// TIA Portal V20 export
TYPE "OPC_DestRequest_Ack"
// stored: Namespace ProductionLine
   STRUCT
      AckSeq : Int;   // //Communication flag, described in the Request - Response tab
      DecisionPoint : String[30];   // // Machine/workstation code:- DP1,…, DP4
      Barcode : String[30];   // // Unique identification of scanned KLTs. For NoRead use ??????????
      State : String[10];   // // Response status: - OK = task ready - NG (not good) = error
      Destination : String[30];   // Identification of the target location: - IP1...IP9
      ErrorReason : String[150];   // // Reason for error in case of status = NG.
   END_STRUCT;
END_TYPE
